// TwinCAT 3 PLC project OOPS_Interface
// ProgramVersion: 3.1.4026.17
// CompilerDefines: VISU_USEPROPERTYINFO
// libraries:
//   Tc2_Standard, * (Beckhoff Automation GmbH)
//   Tc2_System, * (Beckhoff Automation GmbH)
//   VisuSymbols, 4.5.0.0 (System)
// project tree:
//   DUTs/ ET_ResultShiftRegister.TcDUT
//   / GlobalTextList.TcGTLO, PlcTask.TcTTO, Visualization Manager.TcVMO (not stored)
//   POUs/ FB_FIFO_OOP.TcPOU, MAIN.TcPOU, SR_FIFO.TcPOU
//   POUs/FIFO_Props_Itfs/ FB_FIFO.TcPOU, FB_FIFO_1.TcPOU
//   POUs/Push and Pick Using Interface/ FB_Picker_Itf.TcPOU, FB_Pusher_Itf.TcPOU, IF_EmptyRegister.TcIO, IF_FillRegister.TcIO, IF_Register.TcIO, SR_Push_and_pick_ITF.TcPOU
//   VISUs/ Visualization.TcVIS

CONFIGURATION OOPS_Interface
    RESOURCE PLC ON TwinCAT3
        TASK PlcTask(INTERVAL := T#10ms, PRIORITY := 20);
        PROGRAM MAIN WITH PlcTask : MAIN;
        PROGRAM SR_FIFO WITH PlcTask : SR_FIFO;
    END_RESOURCE
END_CONFIGURATION

// ---- DUTs/ET_ResultShiftRegister.TcDUT
{attribute 'qualified_only'}
{attribute 'strict'}
{attribute 'to_string'}
TYPE ET_ResultShiftRegister :
(
	NotInitialised,
	LengthInvalid,
	PositionIsWrong,
	InitDone,
	RegNumberInvalid,
	GetDone,
	PutDone,
	ErrorQuitDone,
	RegisterIsEmpty,
	RegisterISFull,
	OverwriteDone,
	ReadRegisterDone
	
);
END_TYPE

// ---- POUs/Push and Pick Using Interface/IF_EmptyRegister.TcIO
INTERFACE IF_EmptyRegister EXTENDS __SYSTEM.IQueryInterface

METHOD Get : DINT
VAR_INPUT
END_VAR
END_METHOD

PROPERTY xReadyForGet : BOOL
GET
END_GET
END_PROPERTY

END_INTERFACE

// ---- POUs/Push and Pick Using Interface/IF_FillRegister.TcIO
INTERFACE IF_FillRegister EXTENDS __SYSTEM.IQueryInterface

METHOD put : BOOL
VAR_INPUT
	i_diInValue : DINT;
END_VAR
END_METHOD

PROPERTY xReadyForPut : BOOL
GET
END_GET
END_PROPERTY

END_INTERFACE

// ---- POUs/Push and Pick Using Interface/IF_Register.TcIO
INTERFACE IF_Register EXTENDS _SYSTEM.IQueryInterface

PROPERTY adiRegister : REFERENCE TO ARRAY[1..8] OF DINT
GET
END_GET
END_PROPERTY

PROPERTY PUBLIC etResult : ET_ResultShiftRegister
GET
END_GET
END_PROPERTY

END_INTERFACE

// ---- POUs/MAIN.TcPOU
PROGRAM MAIN
VAR
 
END_VAR

END_PROGRAM

// ---- POUs/SR_FIFO.TcPOU
PROGRAM SR_FIFO
VAR
	fbFiFO : FB_FIFO_OOP;
	xFirst: BOOL;
	adiRegsiter: ARRAY [1..8] OF DINT;
	iStep: INT;
	diOutValue : DINT;
END_VAR

adiRegsiter := fbFIFO.adiRegister;
CASE iStep OF 
	
	10:fbFIFO.Init(-1);
	
	20: IF fbFIFO.xReadyForPut THEN
			fbFIFO.Put(23);
		END_IF
	
	30: IF fbFIFO.xReadyForGet THEN
			diOutValue:=fbFIFO.Get();
		END_IF
	
	
END_CASE
iStep:=0;

ACTION RandomGenerator:

END_ACTION

END_PROGRAM

// ---- POUs/FB_FIFO_OOP.TcPOU
FUNCTION_BLOCK FB_FIFO_OOP IMPLEMENTS IF_EmptyRegister
VAR
	adiRegsiter_local   	: ARRAY[1..8] OF DINT;
	i  						: INT ;
	diRegisterLocalValue 	: DINT;
	diNumberofElements_Local 		: DINT;
	etResult_Local			: ET_ResultShiftRegister;
	xReadyforPut_Local		: BOOL:=TRUE;
	xReadyforGet_Local       : BOOL;
	diInitValue_loc         :DINT;
	diLastRegisterValue     :DINT;	
END_VAR

PROPERTY adiRegister : REFERENCE TO ARRAY[1..8] OF DINT
GET
adiRegister REF= THIS^.adiRegsiter_local;
END_GET
END_PROPERTY

PROPERTY etResult : ET_ResultShiftRegister
GET
etResult :=THIS^.etResult_Local;
END_GET
END_PROPERTY

METHOD Get : DINT
VAR_INPUT
END_VAR
Get := THIS^.adiRegsiter_local[diNumberofElements_Local];
THIS^.diLastRegisterValue := Get;

THIS^.adiRegsiter_local[diNumberofElements_Local] :=THIS^.diInitValue_loc;
THIS^.diNumberofElements_Local:=THIS^.diNumberofElements_Local-1;
THIS^.etResult_Local:= ET_ResultShiftRegister.GetDone;
THIS^.xReadyforPut_Local := TRUE;	

IF diNumberofElements_Local= 0 THEN
	THIS^.etResult_Local:= ET_ResultShiftRegister.RegisterIsEmpty;
	THIS^.xReadyforGet_Local:= FALSE;
END_IF
END_METHOD

METHOD PUBLIC Init : BOOL
VAR_INPUT
	i_diInitValue : DINT;
END_VAR
VAR
	i : INT;
END_VAR

FOR i :=  1 TO 8 DO 
	THIS^.adiRegsiter_local[i]:= i_diInitValue;
END_FOR
THIS^.etResult_Local:= ET_ResultShiftRegister.InitDone;

THIS^.xReadyforPut_Local:=TRUE;
THIS^.xReadyforGet_Local:=FALSE;

THIS^.diInitValue_loc := i_diInitValue;
END_METHOD

METHOD Put : DINT
VAR_INPUT
	i_diInValue : DINT;
END_VAR
IF THIS^.diNumberofElements_Local<8 THEN
	THIS^.diNumberofElements_Local:= THIS^.diNumberofElements_Local+1 ;
	FOR i:=8 TO 2 BY -1 DO 
		THIS^.adiRegsiter_local[i]:=THIS^.adiRegsiter_local[i-1];		
	END_FOR
	THIS^.adiRegsiter_local[1]:=i_diInValue;
	THIS^.etResult_Local:= ET_ResultShiftRegister.PutDone;
	THIS^.xReadyforGet_Local := TRUE;
END_IF
IF THIS^.diNumberofElements_Local=8 THEN
		THIS^.etResult_Local:= ET_ResultShiftRegister.RegisterISFull;
		THIS^.xReadyforPut_Local := FALSE;	
END_IF
END_METHOD

PROPERTY xReadyForGet : BOOL
GET
xReadyForGet := THIS^.xReadyforGet_Local;
END_GET
END_PROPERTY

PROPERTY xReadyForPut : BOOL
GET
xReadyForPut := THIS^.xReadyforPut_Local;
END_GET
END_PROPERTY

END_FUNCTION_BLOCK

// ---- POUs/FIFO_Props_Itfs/FB_FIFO.TcPOU
FUNCTION_BLOCK FB_FIFO
VAR_INPUT
END_VAR
VAR_OUTPUT
END_VAR
VAR
	fbfifo : FB_FIFO_OOP;
END_VAR

//FB_Init is always available implicitly and it is used primarily for initialization.
//The return value is not evaluated. For a specific influence, you can also declare the
//methods explicitly and provide additional code there with the standard initialization
//code. You can evaluate the return value.
METHOD FB_Init: BOOL
VAR_INPUT
    bInitRetains: BOOL; // TRUE: the retain variables are initialized (reset warm / reset cold)
    bInCopyCode: BOOL;  // TRUE: the instance will be copied to the copy code afterward (online change)   
END_VAR
THIS^.fbfifo.Init(-3);
END_METHOD

PROPERTY ifEmptyRegister : IF_EmptyRegister
GET
ifEmptyRegister :=THIS^.fbfifo;
END_GET
END_PROPERTY

PROPERTY ifFillRegister : IF_FillRegister
GET
ifEmptyRegister := THIS^.ifFillRegister;
END_GET
END_PROPERTY

PROPERTY ifRegister : IF_Register
GET
ifRegister:=THIS^.fbfifo;
END_GET
END_PROPERTY

END_FUNCTION_BLOCK

// ---- POUs/FIFO_Props_Itfs/FB_FIFO_1.TcPOU
FUNCTION_BLOCK FB_FIFO_1 EXTENDS FB_FIFO_OOP
VAR_INPUT
END_VAR
VAR_OUTPUT
END_VAR
VAR
END_VAR

PROPERTY ifEmptyRegister : IF_EmptyRegister
GET
ifEmptyRegister:=super^;
END_GET
END_PROPERTY

PROPERTY ifFillRegister : IF_FillRegister
GET
ifFillRegister:=super^;
END_GET
END_PROPERTY

PROPERTY ifRegister : IF_Register
GET
ifRegister:=super^;
END_GET
END_PROPERTY

END_FUNCTION_BLOCK

// ---- POUs/Push and Pick Using Interface/FB_Picker_Itf.TcPOU
FUNCTION_BLOCK FB_Picker_Itf
VAR_INPUT
	i_ifEmptyRegister :IF_EmptyRegister;
END_VAR
VAR_OUTPUT
	diProductNr : DINT;
END_VAR
VAR_IN_OUT
	iq_xSensor : BOOL;
END_VAR

IF i_ifEmptyRegister<> 0 THEN
	IF iq_xSensor AND i_ifEmptyRegister.xReadyForGet THEN
		iq_xSensor:= FALSE;
		diProductNr:=i_ifEmptyRegister.Get();
	END_IF
	
END_IF

END_FUNCTION_BLOCK

// ---- POUs/Push and Pick Using Interface/FB_Pusher_Itf.TcPOU
FUNCTION_BLOCK FB_Pusher_Itf
VAR_INPUT
	i_ifRegister : IF_Register;
	
END_VAR
VAR_OUTPUT
END_VAR
VAR
	diProductCounter : DINT;
	ifFillRegister : IF_FillRegister;
	
	xSucess: BOOL;
END_VAR

VAR_IN_OUT
	iq_xSensor: BOOL;
END_VAR

xSucess :=__QUERYINTERFACE(i_ifRegister,ifFillRegister);
IF xSucess THEN
	diProductCounter := diProductCounter+1;
	IF iq_xSensor AND ifFillRegister.xReadyForPut THEN
		iq_xSensor:=FALSE;
		ifFillRegister.put(i_diInValue:=diProductCounter);
	END_IF
END_IF

END_FUNCTION_BLOCK

// ---- POUs/Push and Pick Using Interface/SR_Push_and_pick_ITF.TcPOU
PROGRAM SR_Push_and_pick_ITF
VAR
	fbFIFO : FB_FIFO_OOP;
	fbPusher : FB_Pusher_Itf;
	xPush  : BOOL;
	fbPicker  : FB_Picker_Itf;
	xPick  : BOOL;
END_VAR

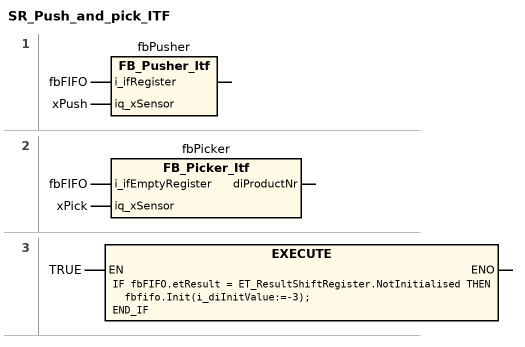
// NETWORK 1
fbPusher(i_ifRegister := fbFIFO, iq_xSensor := xPush); // FB_Pusher_Itf

// NETWORK 2
fbPicker(i_ifEmptyRegister := fbFIFO, iq_xSensor := xPick); // FB_Picker_Itf

// NETWORK 3
IF fbFIFO.etResult = ET_ResultShiftRegister.NotInitialised THEN
	fbfifo.Init(i_diInitValue:=-3);
END_IF

END_PROGRAM

// ---- VISUs/Visualization.TcVIS
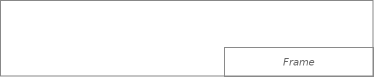
VISUALIZATION Visualization  // 374x77
    Frame (224,47 150x30)
END_VISUALIZATION
